{attribute 'Tc2GvlVarNames'}
VAR_CONFIG
	.Dali_K522A1_DALI_IN AT %IB253		 : ST_DALIV2InData;
	.Dali_K522A1_DALI_OUT AT %QB141 		: ST_DALIV2OutData;
END_VAR

(* stored: Version 1.1.0.1, ProductVersion 3.1.4024.10
   GVL Variablen_Konfiguration: Id {418cb1f7-448c-4913-b972-128724ec2bc0} *)
